(* Logix 5000 project; controller Reto1 vendor 1 type 14 code 156 rev 30.11; software revision 30.00 *)

TASK MainTask (continuous, watchdog 500 ms) : MainProgram

MODULES
   Local : vendor 1 type 14 code 156 (Compact 0, rev 30.11)
      DI_4 : 1769-IQ16 (Compact 4, rev 1.1, Input RPI 20 ms)
      DO_5 : vendor 1 type 7 code 86 (Compact 5, rev 2.1, Output RPI 20 ms)
END_MODULES

VAR_GLOBAL   (* controller tags *)
   Bot_Start : BOOL;
   Bot_Stop : BOOL;
   C0 : BOOL;   // OK_INITIALIZATION
   C1 : BOOL;   // OK_STSTEM_ON
   C2 : BOOL;   // OK_POS_TAPA
   C3 : BOOL;   // OK_POS_BASE
   C4 : BOOL;   // OK_FORMADO
   C5 : BOOL;   // OK_FORMADO2
   C6 : BOOL;   // OK_RESET_PROCESS
   CONT_CAJAS : COUNTER := (PRE := 10);
   CONT_INT : INT;
   E0 : BOOL;   // INITIALIZATION
   E1 : BOOL;   // STSTEM_ON
   E2 : BOOL;   // POS_TAPA
   E3 : BOOL;   // POS_BASE
   E4 : BOOL;   // FORMADO
   E5 : BOOL;   // FORMADO2
   E6 : BOOL;   // RESET_PROCESS
   ENT_BASE : BOOL;
   ENT_LID : BOOL;
   ES : BOOL;   // Help Emergency Stop
   GD_IN_0 : BOOL;   // GD_MOVING_X
   GD_IN_1 : BOOL;   // GD_MOVING_Z
   GD_IN_10 : BOOL;   // START_ALL
   GD_IN_11 : BOOL;   // RESET
   GD_IN_12 : BOOL;   // STOP_ALL
   GD_IN_13 : BOOL;   // GD Emergency Stop
   GD_IN_2 : BOOL;   // ITEM_DETECTER
   GD_IN_3 : BOOL;   // LID_AT_PLACE
   GD_IN_4 : BOOL;   // GD_LID_CLAMPED
   GD_IN_5 : BOOL;   // POS_LIMIT_LIDS
   GD_IN_6 : BOOL;   // BASE_AT_PLACE
   GD_IN_7 : BOOL;   // GD_BASE_CLAMPED
   GD_IN_8 : BOOL;   // POS_LIMIT_BASES
   GD_IN_9 : BOOL;   // GD_PART_LEAVING
   GD_OUT_0 : BOOL;   // MOVE_X
   GD_OUT_1 : BOOL;   // MOVE_Z
   GD_OUT_10 : BOOL;   // RESET_LIGHT
   GD_OUT_11 : BOOL;   // STOP_LIGHT
   GD_OUT_2 : BOOL;   // GRAB
   GD_OUT_3 : BOOL;   // LIDS_CONVEYOR
   GD_OUT_4 : BOOL;   // CLAMP_LID
   GD_OUT_5 : BOOL;   // GD_LID_POS_RAISED
   GD_OUT_6 : BOOL;   // BASES_CONVEYOR
   GD_OUT_7 : BOOL;   // CLAMP_BASE
   GD_OUT_8 : BOOL;   // GD_BASE_POS_RAISED
   GD_OUT_9 : BOOL;   // START_LIGHT
   INT1 : BOOL;   // INT1
   INT_OUT_0 : INT;
   OK_RESET : BOOL;
   ONS_E2 : BOOL;
   ONS_E3 : BOOL;
   ONS_GRAB_OFF : BOOL;
   ONS_INIT_E4 : BOOL;
   ONS_ITEM_DETECTED : BOOL;
   ONS_MX : BOOL;
   ONS_MZ2 : BOOL;
   ONS_OK_FORMADO : BOOL;
   OSF_BASE_IN : BOOL;
   OSF_BASE_OUT : BOOL;
   OSF_BASE_RAISED_ON : BOOL;
   OSF_BASE_RAISED_OUT : BOOL;
   OSF_GRAB_IN : BOOL;
   OSF_GRAB_OUT : BOOL;
   OSF_LID_IN : BOOL;
   OSF_LID_OUT : BOOL;
   OSR_FORMADO_IN : BOOL;
   OSR_FORMADO_OUT : BOOL;
   OSR_GRAB_IN : BOOL;
   OSR_GRAB_OFF : BOOL;
   P1 : BOOL;   // TOGGLE BIT
   PC_GOFF : BOOL;
   PC_HZ1 : BOOL;
   PC_HZ2 : BOOL;
   PC_MX : BOOL;
   PS_MOTOR : ALIAS FOR Local:5:O.Data.0;
   PS_START : ALIAS FOR Local:4:I.Data.1;
   PS_STOP : ALIAS FOR Local:4:I.Data.0;
   TB : BOOL;   // TOGGLE_BIT
   TB1 : BOOL;
   TB2 : BOOL;
   TB_E2 : BOOL;
   TB_GRAB : BOOL;
   TB_GRAB_OFF : BOOL;
   TB_HX : BOOL;
   TB_HZ : BOOL;
   TB_HZ_2 : BOOL;
   TB_X : BOOL;
   TB_Z1 : BOOL;
   TB_Z2 : BOOL;
   TIMER_GRAB_OFF : TIMER := (PRE := 250);
   TIMER_HX : TIMER := (PRE := 250);
   TIMER_MZ2 : TIMER := (PRE := 250);
   TIMER_OK_FORMADO : TIMER := (PRE := 250);
   TON_BASE : TIMER := (PRE := 100);
   TON_IE4 : TIMER := (PRE := 500);
   TON_LEAVING : TIMER := (PRE := 500);
   TON_LID : TIMER := (PRE := 100);
END_VAR

PROGRAM MainProgram   (* main routine MainRoutine *)

ROUTINE A_SETUP   (* ladder *)
   0 (stored rung type 13): ;
END_ROUTINE

ROUTINE A_SETUP1   (* ladder *)
   0 (stored rung type 13): ;
END_ROUTINE

ROUTINE B_PREPARING   (* ladder *)
   0 (stored rung type 13): ;
END_ROUTINE

ROUTINE C_FORMING   (* ladder *)
END_ROUTINE

ROUTINE MainRoutine   (* ladder *)
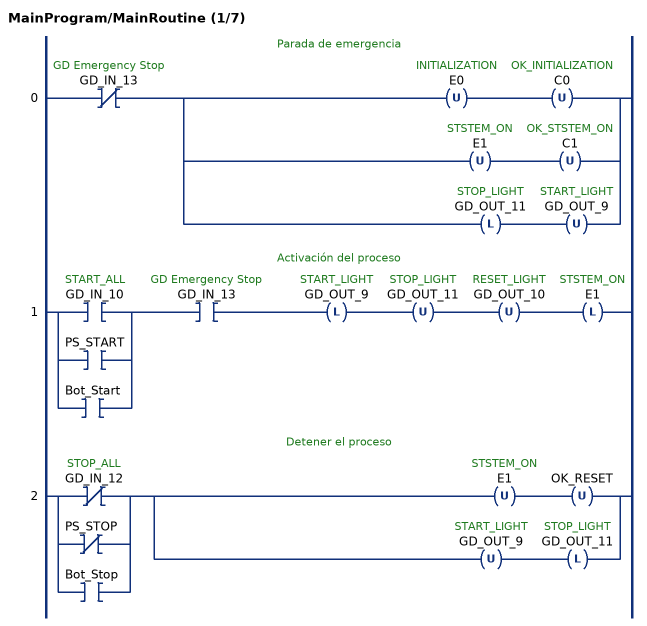
   // Parada de emergencia
   0: XIO(GD_IN_13)[OTU(E0) OTU(C0) ,[OTU(E1) OTU(C1) ,OTL(GD_OUT_11) OTU(GD_OUT_9) ] ];
   // Activación del proceso
   1: [XIC(GD_IN_10) ,[XIC(PS_START) ,XIC(Bot_Start) ] ]XIC(GD_IN_13)OTL(GD_OUT_9)OTU(GD_OUT_11)OTU(GD_OUT_10)OTL(E1);
   // Detener el proceso
   2: [XIO(GD_IN_12) ,[XIO(PS_STOP) ,XIC(Bot_Stop) ] ][OTU(E1) OTU(OK_RESET) ,OTU(GD_OUT_9) OTL(GD_OUT_11) ];
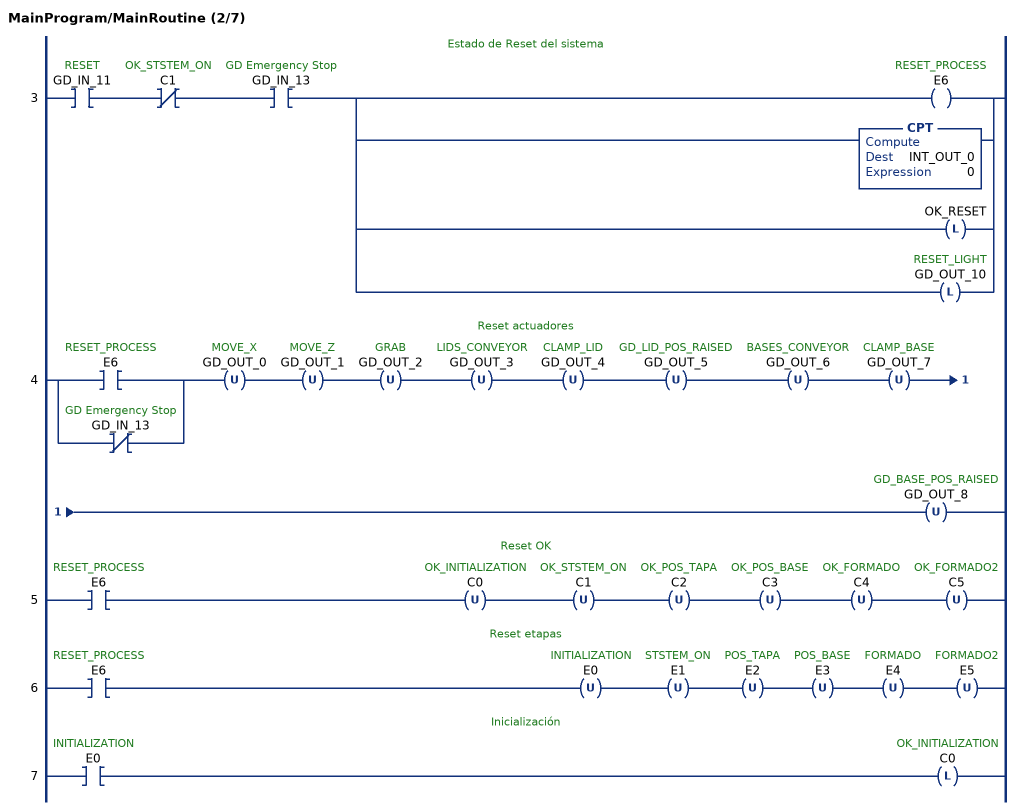
   // Estado de Reset del sistema
   3: XIC(GD_IN_11)XIO(C1)XIC(GD_IN_13)[OTE(E6) ,[CPT(INT_OUT_0,0) ,[OTL(OK_RESET) ,OTL(GD_OUT_10) ] ] ];
   // Reset actuadores
   4: [XIC(E6) ,XIO(GD_IN_13) ]OTU(GD_OUT_0)OTU(GD_OUT_1)OTU(GD_OUT_2)OTU(GD_OUT_3)OTU(GD_OUT_4)OTU(GD_OUT_5)OTU(GD_OUT_6)OTU(GD_OUT_7)OTU(GD_OUT_8);
   // Reset OK
   5: XIC(E6)OTU(C0)OTU(C1)OTU(C2)OTU(C3)OTU(C4)OTU(C5);
   // Reset etapas
   6: XIC(E6)OTU(E0)OTU(E1)OTU(E2)OTU(E3)OTU(E4)OTU(E5);
   // Inicialización
   7: XIC(E0)OTL(C0);
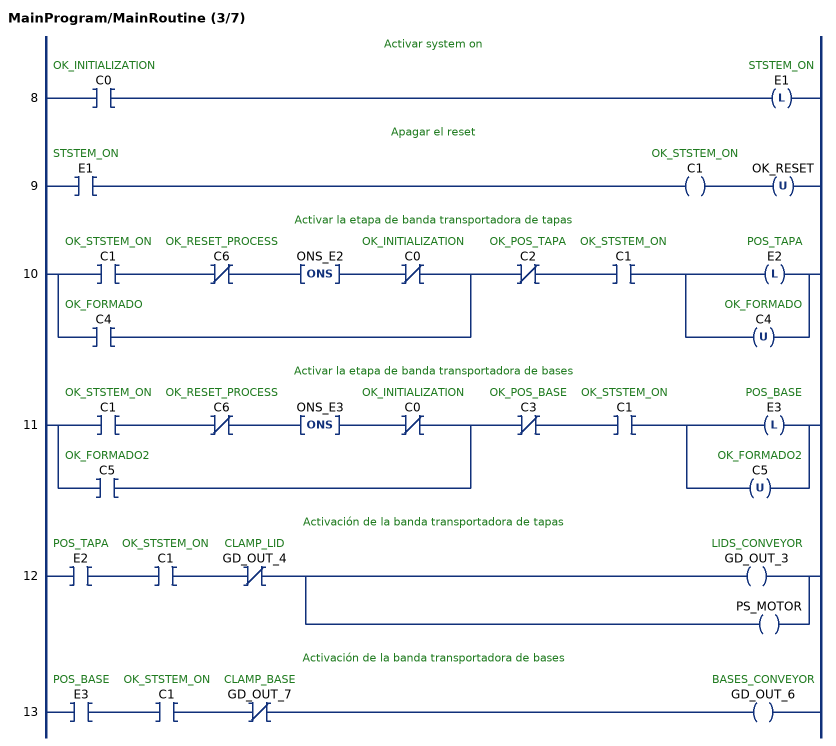
   // Activar system on
   8: XIC(C0)OTL(E1);
   // Apagar el reset
   9: XIC(E1)OTE(C1)OTU(OK_RESET);
   // Activar la etapa de banda transportadora de tapas
   10: [XIC(C1) XIO(C6) ONS(ONS_E2) XIO(C0) ,XIC(C4) ]XIO(C2)XIC(C1)[OTL(E2) ,OTU(C4) ];
   // Activar la etapa de banda transportadora de bases
   11: [XIC(C1) XIO(C6) ONS(ONS_E3) XIO(C0) ,XIC(C5) ]XIO(C3)XIC(C1)[OTL(E3) ,OTU(C5) ];
   // Activación de la banda transportadora de tapas
   12: XIC(E2)XIC(C1)XIO(GD_OUT_4)[OTE(GD_OUT_3) ,OTE(PS_MOTOR) ];
   // Activación de la banda transportadora de bases
   13: XIC(E3)XIC(C1)XIO(GD_OUT_7)OTE(GD_OUT_6);
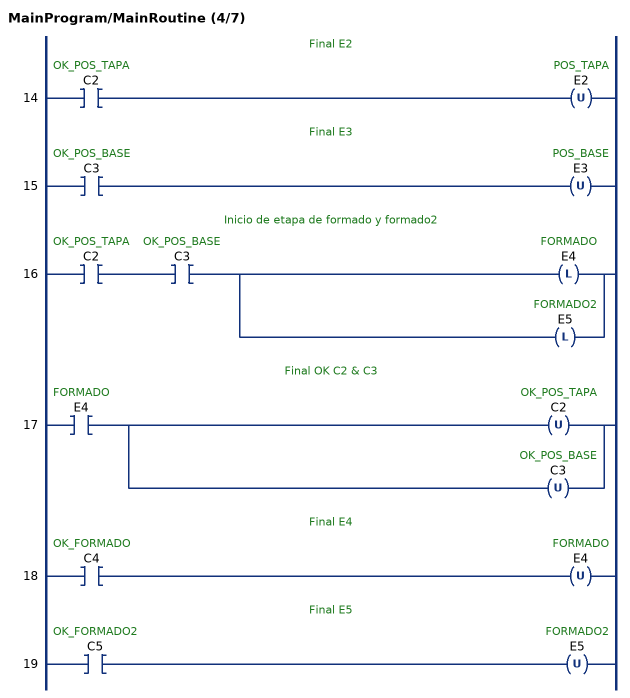
   // Final E2
   14: XIC(C2)OTU(E2);
   // Final E3
   15: XIC(C3)OTU(E3);
   // Inicio de etapa de formado y formado2
   16: XIC(C2)XIC(C3)[OTL(E4) ,OTL(E5) ];
   // Final OK C2 & C3
   17: XIC(E4)[OTU(C2) ,OTU(C3) ];
   // Final E4
   18: XIC(C4)OTU(E4);
   // Final E5
   19: XIC(C5)OTU(E5);
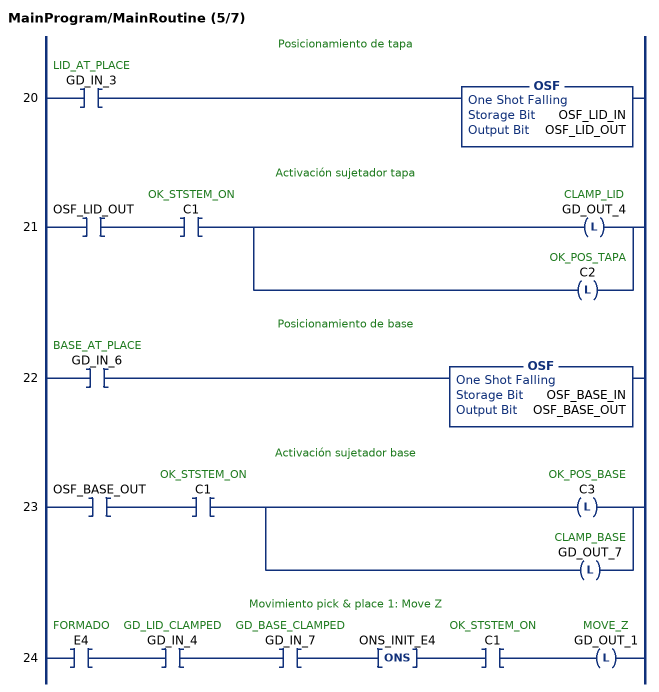
   // Posicionamiento de tapa
   20: XIC(GD_IN_3)OSF(OSF_LID_IN,OSF_LID_OUT);
   // Activación sujetador tapa
   21: XIC(OSF_LID_OUT)XIC(C1)[OTL(GD_OUT_4) ,OTL(C2) ];
   // Posicionamiento de base
   22: XIC(GD_IN_6)OSF(OSF_BASE_IN,OSF_BASE_OUT);
   // Activación sujetador base
   23: XIC(OSF_BASE_OUT)XIC(C1)[OTL(C3) ,OTL(GD_OUT_7) ];
   // Movimiento pick & place 1: Move Z
   24: XIC(E4)XIC(GD_IN_4)XIC(GD_IN_7)ONS(ONS_INIT_E4)XIC(C1)OTL(GD_OUT_1);
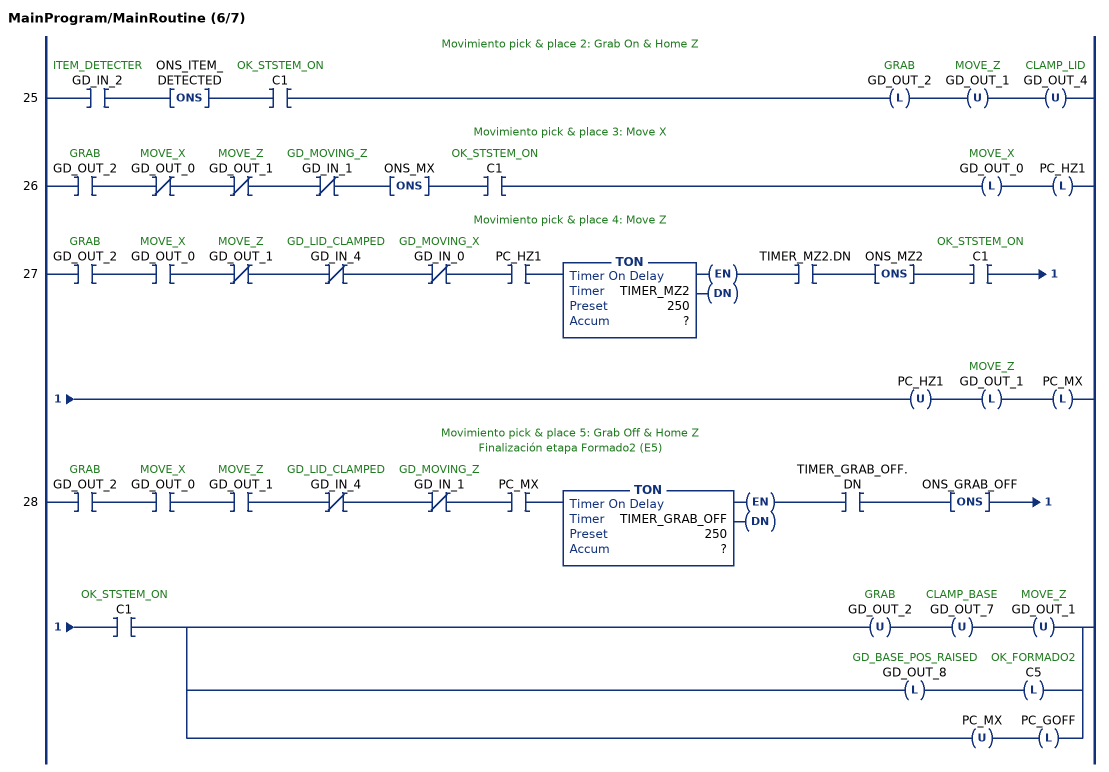
   // Movimiento pick & place 2: Grab On & Home Z
   25: XIC(GD_IN_2)ONS(ONS_ITEM_DETECTED)XIC(C1)OTL(GD_OUT_2)OTU(GD_OUT_1)OTU(GD_OUT_4);
   // Movimiento pick & place 3: Move X
   26: XIC(GD_OUT_2)XIO(GD_OUT_0)XIO(GD_OUT_1)XIO(GD_IN_1)ONS(ONS_MX)XIC(C1)OTL(GD_OUT_0)OTL(PC_HZ1);
   // Movimiento pick & place 4: Move Z
   27: XIC(GD_OUT_2)XIC(GD_OUT_0)XIO(GD_OUT_1)XIO(GD_IN_4)XIO(GD_IN_0)XIC(PC_HZ1)TON(TIMER_MZ2,?,?)XIC(TIMER_MZ2.DN)ONS(ONS_MZ2)XIC(C1)OTU(PC_HZ1)OTL(GD_OUT_1)OTL(PC_MX);
   // Movimiento pick & place 5: Grab Off & Home Z
   // Finalización etapa Formado2 (E5)
   28: XIC(GD_OUT_2)XIC(GD_OUT_0)XIC(GD_OUT_1)XIO(GD_IN_4)XIO(GD_IN_1)XIC(PC_MX)TON(TIMER_GRAB_OFF,?,?)XIC(TIMER_GRAB_OFF.DN)ONS(ONS_GRAB_OFF)XIC(C1)[OTU(GD_OUT_2) OTU(GD_OUT_7) OTU(GD_OUT_1) ,[OTL(GD_OUT_8) OTL(C5) ,OTU(PC_MX) OTL(PC_GOFF) ] ];
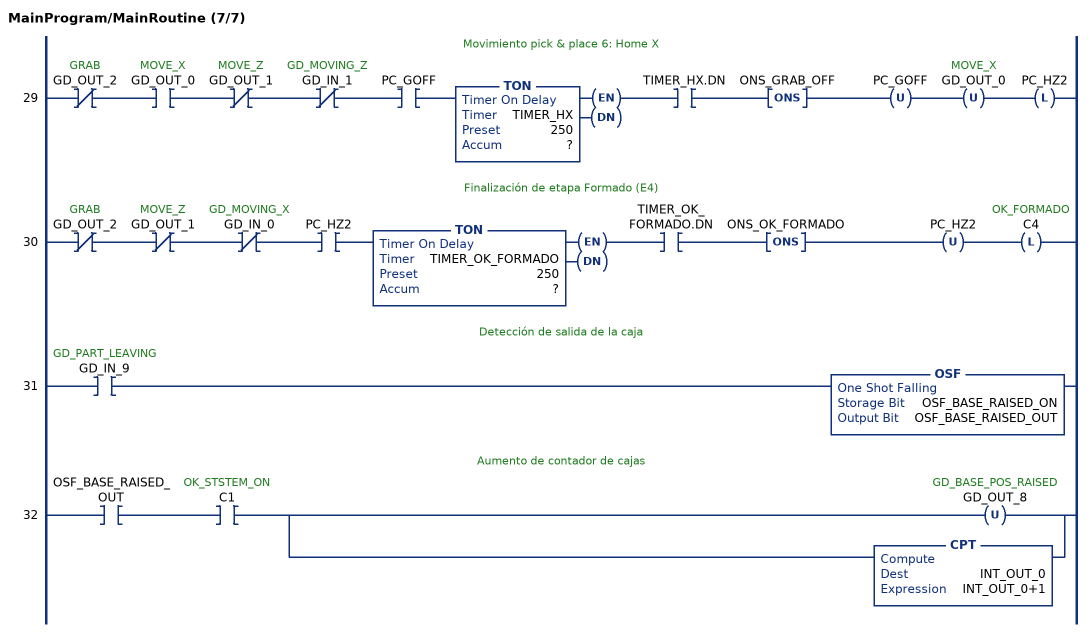
   // Movimiento pick & place 6: Home X
   29: XIO(GD_OUT_2)XIC(GD_OUT_0)XIO(GD_OUT_1)XIO(GD_IN_1)XIC(PC_GOFF)TON(TIMER_HX,?,?)XIC(TIMER_HX.DN)ONS(ONS_GRAB_OFF)OTU(PC_GOFF)OTU(GD_OUT_0)OTL(PC_HZ2);
   // Finalización de etapa Formado (E4)
   30: XIO(GD_OUT_2)XIO(GD_OUT_1)XIO(GD_IN_0)XIC(PC_HZ2)TON(TIMER_OK_FORMADO,?,?)XIC(TIMER_OK_FORMADO.DN)ONS(ONS_OK_FORMADO)OTU(PC_HZ2)OTL(C4);
   // Detección de salida de la caja
   31: XIC(GD_IN_9)OSF(OSF_BASE_RAISED_ON,OSF_BASE_RAISED_OUT);
   // Aumento de contador de cajas
   32: XIC(OSF_BASE_RAISED_OUT)XIC(C1)[OTU(GD_OUT_8) ,CPT(INT_OUT_0,INT_OUT_0+1) ];
END_ROUTINE

ROUTINE RESET   (* ladder *)
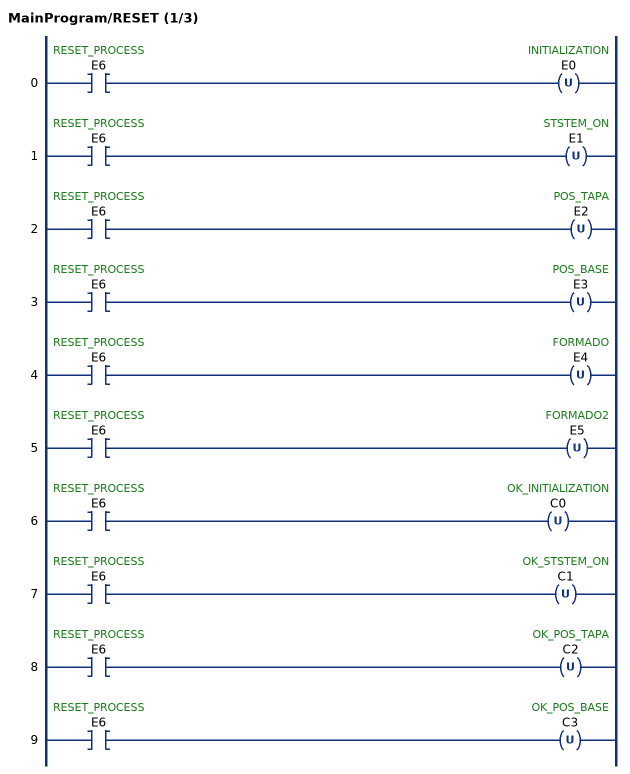
   0: XIC(E6)OTU(E0);
   1: XIC(E6)OTU(E1);
   2: XIC(E6)OTU(E2);
   3: XIC(E6)OTU(E3);
   4: XIC(E6)OTU(E4);
   5: XIC(E6)OTU(E5);
   6: XIC(E6)OTU(C0);
   7: XIC(E6)OTU(C1);
   8: XIC(E6)OTU(C2);
   9: XIC(E6)OTU(C3);
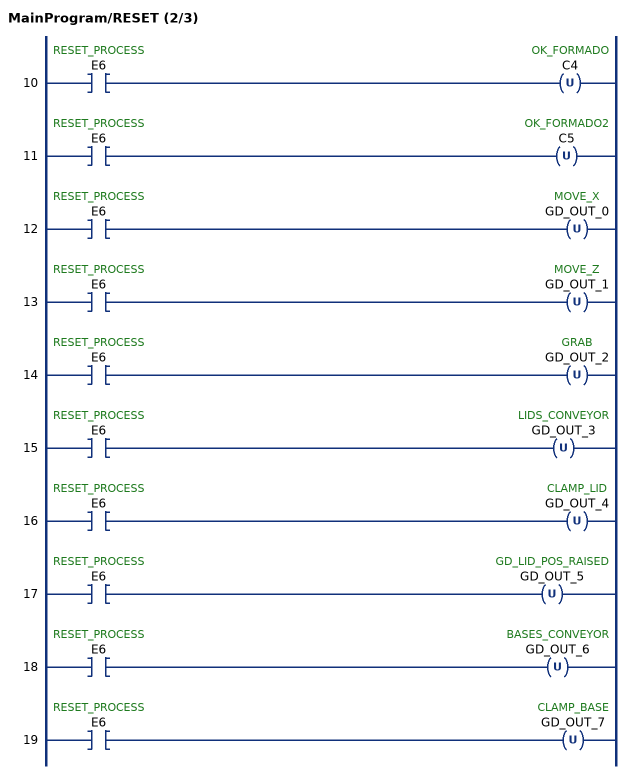
   10: XIC(E6)OTU(C4);
   11: XIC(E6)OTU(C5);
   12: XIC(E6)OTU(GD_OUT_0);
   13: XIC(E6)OTU(GD_OUT_1);
   14: XIC(E6)OTU(GD_OUT_2);
   15: XIC(E6)OTU(GD_OUT_3);
   16: XIC(E6)OTU(GD_OUT_4);
   17: XIC(E6)OTU(GD_OUT_5);
   18: XIC(E6)OTU(GD_OUT_6);
   19: XIC(E6)OTU(GD_OUT_7);
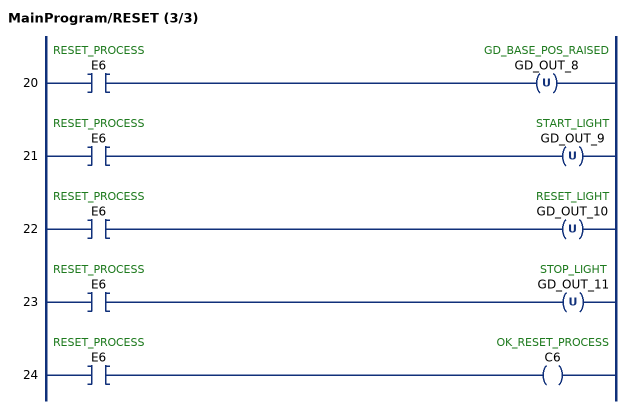
   20: XIC(E6)OTU(GD_OUT_8);
   21: XIC(E6)OTU(GD_OUT_9);
   22: XIC(E6)OTU(GD_OUT_10);
   23: XIC(E6)OTU(GD_OUT_11);
   24: XIC(E6)OTE(C6);
END_ROUTINE
END_PROGRAM
